// TwinCAT 3 PLC project Oefeningen3_
// ProgramVersion: 3.1.4024.0
// libraries:
//   Tc2_BABasic, * (Beckhoff Automation GmbH)
//   Tc2_Standard, * (Beckhoff Automation GmbH)
//   Tc2_System, * (Beckhoff Automation GmbH)
//   Tc2_Utilities, * (Beckhoff Automation GmbH)
//   Tc3_Module, * (Beckhoff Automation GmbH)
// project tree:
//   DUTs/ Pers_data.TcDUT
//   / GlobalTextList.TcGTLO, PlcTask.TcTTO, Visualization Manager.TcVMO (not stored)
//   POUs/ CheckBounds.TcPOU, CheckRangeInt.TcPOU, FB_Click_Log.TcPOU, FB_DrukknopSpecial.TcPOU, FB_GetMinimum.TcPOU, FB_PWM.TcPOU, FB_SearchString.TcPOU, FGetMinimum.TcPOU, MAIN.TcPOU, prg_Click_Log.TcPOU, prg_Druktoets_Functies.TcPOU, prg_GetMinimum.TcPOU, prg_Personeelsdata.TcPOU, prg_PWM.TcPOU, prg_SearchString.TcPOU
//   VISUs/ Visualization_Click_Logger.TcVIS, Visualization_GetMinimumClicker.TcVIS
// (motion and I/O tree: see PLC project oefeningen1)
// real-time tasks:
//   TASK PlcTask: cycle T#10ms, priority 20, ADS port 350
//   TASK PlcTask1: cycle T#10ms, priority 21, ADS port 351
//   TASK PlcTask2: cycle T#10ms, priority 22, ADS port 352
//   TASK PlcTask3: cycle T#10ms, priority 23, ADS port 353
//   TASK PlcTask4: cycle T#10ms, priority 24, ADS port 354

CONFIGURATION Oefeningen3_
    RESOURCE PLC ON TwinCAT3
        TASK PlcTask(INTERVAL := T#10ms, PRIORITY := 24);
        PROGRAM MAIN WITH PlcTask : MAIN;
    END_RESOURCE
END_CONFIGURATION

// ---- DUTs/Pers_data.TcDUT
TYPE Pers_data :
STRUCT
	Name      : STRING(25);
	Firstname : STRING(25);
	Age       : INT;
	Address   : STRING(55);
END_STRUCT
END_TYPE

// ---- POUs/MAIN.TcPOU
PROGRAM MAIN
VAR
END_VAR

//prg_PWM();
//prg_Click_Log();
//prg_GetMinimum();
//prg_Personeelsdata();
//prg_SearchString();
prg_Druktoets_Functies();

END_PROGRAM

// ---- POUs/prg_Druktoets_Functies.TcPOU
PROGRAM prg_Druktoets_Functies
VAR
	FB_Drukknop_Special: FB_DrukknopSpecial;
END_VAR

FB_Drukknop_Special(bDrukknop:= , bSingle=> , bDouble=> , bLong=> );

END_PROGRAM

// ---- POUs/FB_DrukknopSpecial.TcPOU
FUNCTION_BLOCK FB_DrukknopSpecial
VAR_INPUT
    bDrukknop : BOOL;          // fysiek knopsignaal
END_VAR

VAR_OUTPUT
    bSingle    : BOOL;
    bDouble    : BOOL;
    bLong      : BOOL;
END_VAR

VAR
    fbSD : FB_SingleDoubleClick;
    fbSL : FB_ShortLongClick;
END_VAR

// --- Doorgeven van de knop als input ---
fbSD(bSwitch := bDrukknop, tSwitchTime := T#500MS);
fbSL(bSwitch := bDrukknop, tSwitchTime := T#1S);

// --- Outputs ---
bSingle := fbSD.bSingleClick AND NOT fbSL.bLongClick;
bDouble := fbSD.bDoubleClick;
bLong   := fbSL.bLongClick;

END_FUNCTION_BLOCK

// ---- POUs/CheckBounds.TcPOU
FUNCTION CheckBounds : INT
VAR_INPUT
    InValue : INT;
END_VAR
VAR
END_VAR

IF InValue < 15 THEN
    CheckBounds := 15;
ELSIF InValue > 24 THEN
    CheckBounds := 24;
ELSE
    CheckBounds := InValue;
END_IF

END_FUNCTION

// ---- POUs/CheckRangeInt.TcPOU
FUNCTION CheckRangeInt : INT
VAR_INPUT
    InValue : INT;
END_VAR
VAR
END_VAR

IF InValue < 0 THEN
    CheckRangeInt := 0;
ELSIF InValue > 32767 THEN
    CheckRangeInt := 32767;
ELSE
    CheckRangeInt := InValue;
END_IF

END_FUNCTION

// ---- POUs/FB_Click_Log.TcPOU
FUNCTION_BLOCK FB_Click_Log
VAR_INPUT
    Drukknop    : BOOL;
END_VAR
VAR_OUTPUT
    Tijden      : ARRAY[1..10] OF TIME;
END_VAR
VAR
    tDrukRegistreren : TP;
    tPauze           : TP;
    FallingTimer     : F_TRIG;
    FallingPauze     : F_TRIG;

    RisingDruk       : R_TRIG;   
    Index            : INT := 0; 
    VorigeET         : TIME := T#0ms;   // nieuwe variabele om vorige tijd op te slaan
	i: INT;
END_VAR

(* Detecteer drukflank *)
RisingDruk(CLK := Drukknop);

(* 5s registratie *)
tDrukRegistreren(IN := Drukknop OR FallingPauze.Q, PT := T#5S);
FallingTimer(CLK := tDrukRegistreren.Q);

(* 2s pauze *)
tPauze(IN := FallingTimer.Q, PT := T#2S);
FallingPauze(CLK := tPauze.Q);

(* reset index na pauze *)
IF FallingPauze.Q THEN
    Index := 0;
    VorigeET := T#0MS;
	FOR i := 1 TO 10 DO
    Tijden[i] := T#0ms;
END_FOR;
END_IF

(* Registreer tijd bij elke drukflank *)
IF RisingDruk.Q AND tDrukRegistreren.Q THEN
    IF Index < 10 THEN
        Index := Index + 1;
        Tijden[Index] := tDrukRegistreren.ET - VorigeET;  // verschil tussen huidige en vorige druk
        VorigeET := tDrukRegistreren.ET;                  // update vorige tijd
    END_IF
END_IF

END_FUNCTION_BLOCK

// ---- POUs/FB_GetMinimum.TcPOU
FUNCTION_BLOCK FB_GetMinimum
VAR_INPUT
	Times : ARRAY[1..10] OF TIME;
END_VAR
VAR_OUTPUT
	MinTime : TIME;
END_VAR
VAR
	i : INT;
END_VAR

(* Initieel minimum = eerste element *)
MinTime := Times[1];

(* Vergelijk met rest van de array *)
FOR i := 2 TO 10 DO
	IF Times[i] < MinTime THEN
		MinTime := Times[i];
	END_IF
END_FOR;

END_FUNCTION_BLOCK

// ---- POUs/FB_PWM.TcPOU
FUNCTION_BLOCK FB_PWM
VAR_INPUT
    Enable     : BOOL;
    Periode    : TIME;   // totale PWM-periode
    DutyCycle  : INT;    // 0 .. 100 (%)
END_VAR

VAR_OUTPUT
    PWM_Out    : BOOL;
END_VAR

VAR
    tPWM       : TON;
    tOn        : TIME;
END_VAR

IF Enable THEN
    (* Bereken ON-tijd *)
    tOn := Periode * DutyCycle / 100;

    tPWM(IN := TRUE, PT := Periode);

    (* PWM-logica *)
    IF tPWM.ET < tOn THEN
        PWM_Out := TRUE;
    ELSE
        PWM_Out := FALSE;
    END_IF

    (* Periode herstarten *)
    IF tPWM.Q THEN
        tPWM(IN := FALSE);
    END_IF
ELSE
    PWM_Out := FALSE;
    tPWM(IN := FALSE);
END_IF

END_FUNCTION_BLOCK

// ---- POUs/FB_SearchString.TcPOU
FUNCTION_BLOCK FB_SearchString
VAR_INPUT
	Person    : Pers_data; //DUT STRUCT
	SearchTxt : STRING(25);
END_VAR
VAR_OUTPUT
	Match     : BOOL;
END_VAR
VAR
	AllText   : STRING(120);
	AllTextLower  : STRING(120);
	SearchLower   : STRING(25);
END_VAR

(* alles samenvoegen *)
AllText := CONCAT(
				CONCAT(Person.Name, Person.Firstname),
				Person.Address
			);

(* naar lowercase omzetten *)
AllTextLower := F_ToLCase(AllText);
SearchLower  := F_ToLCase(SearchTxt);

(* vergelijken *)
IF FIND(AllTextLower, SearchLower) > 0 THEN
	Match := TRUE;
ELSE
	Match := FALSE;
END_IF

END_FUNCTION_BLOCK

// ---- POUs/FGetMinimum.TcPOU
FUNCTION FGetMinimum : TIME
VAR_INPUT
	Times : ARRAY[1..10] OF TIME;
END_VAR
VAR
	i : INT;
	MinVal : TIME;
END_VAR

MinVal := Times[1];

FOR i := 2 TO 10 DO
	IF Times[i] < MinVal THEN
		MinVal := Times[i];
	END_IF
END_FOR;

FGetMinimum := MinVal;

END_FUNCTION

// ---- POUs/prg_Click_Log.TcPOU
PROGRAM prg_Click_Log
VAR	
	ClickLog: FB_Click_Log;

	bDrukknop		AT		%I*		:BOOL;
	LogTijden 		AT		%Q*		:ARRAY[1..10] OF TIME;
END_VAR

ClickLog(Drukknop:= bDrukknop, Tijden=> LogTijden);

END_PROGRAM

// ---- POUs/prg_GetMinimum.TcPOU
PROGRAM prg_GetMinimum
VAR
	FB_GetMinimum: FB_GetMinimum;
	FB_Click_Log: FB_Click_Log;
	bDrukknop		AT		%I*		:BOOL;
	tMinTime		AT		%Q*		:TIME;
	LogTijden 		:ARRAY[1..10] OF TIME;
END_VAR

FB_Click_Log(Drukknop:= bDrukknop, Tijden=> LogTijden);
FB_GetMinimum(Times:= LogTijden, MinTime=> tMinTime);

//Met een functie ipv FunctieBlok (ongetest)
//tMinTime := FGetMinimum(LogTijden);

END_PROGRAM

// ---- POUs/prg_Personeelsdata.TcPOU
PROGRAM prg_Personeelsdata
VAR
	Personeel : ARRAY[1..6] OF Pers_data;
END_VAR

(* P1 *)
Personeel[1].Name      := 'Müller';
Personeel[1].Firstname := 'Peter';
Personeel[1].Age       := 32;
Personeel[1].Address   := 'Postweg 34';

(* P2 *)
Personeel[2].Name      := 'Maesen';
Personeel[2].Firstname := 'Stijn';
Personeel[2].Age       := 15;
Personeel[2].Address   := 'Grote steenweg 8';

(* P3 *)
Personeel[3].Name      := 'Paque';
Personeel[3].Firstname := 'Stéphanie';
Personeel[3].Age       := 42;
Personeel[3].Address   := 'Tongersesteenweg 456';

(* P4 *)
Personeel[4].Name      := 'Fossen';
Personeel[4].Firstname := 'Jo';
Personeel[4].Age       := 20;
Personeel[4].Address   := 'Broekstraat 45';

(* P5 *)
Personeel[5].Name      := 'Poesmans';
Personeel[5].Firstname := 'Benny';
Personeel[5].Age       := 72;
Personeel[5].Address   := 'Veldweg 1A';

(* P6 *)
Personeel[6].Name      := 'Dybek';
Personeel[6].Firstname := 'Isolde';
Personeel[6].Age       := 55;
Personeel[6].Address   := 'Slagerijstraat 6';

END_PROGRAM

// ---- POUs/prg_PWM.TcPOU
PROGRAM prg_PWM
VAR
	PWM: FB_PWM;
	bPWMOUT		AT		%Q*		:BOOL;
END_VAR

PWM(Enable:= TRUE, Periode:= T#1S, DutyCycle:= 25, PWM_Out=> bPWMOUT);

END_PROGRAM

// ---- POUs/prg_SearchString.TcPOU
PROGRAM prg_SearchString
VAR
	Persoon : Pers_data := (
		Name := 'Peeters',
		Firstname := 'Stijn',
		Address := 'Kerkstraat 12'
	);

	SearchFB : FB_SearchString;
	Result   : BOOL;
END_VAR

SearchFB(
	Person := Persoon,
	SearchTxt := 'stijn'
);

Result := SearchFB.Match;

END_PROGRAM

// ---- GlobalTextList.TcGTLO
TEXTLIST GlobalTextList
  841 = 'Drukknop'
END_TEXTLIST

// ---- VISUs/Visualization_Click_Logger.TcVIS
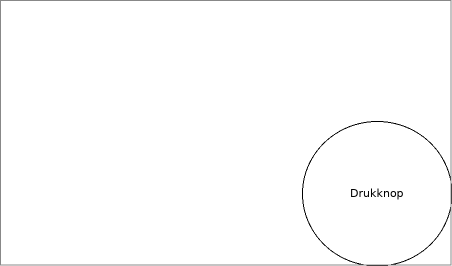
VISUALIZATION Visualization_Click_Logger  // 452x266
    Ellipse (302,121 150x145), "Drukknop"
        tap prg_GetMinimum.bDrukknop
END_VISUALIZATION

// ---- VISUs/Visualization_GetMinimumClicker.TcVIS
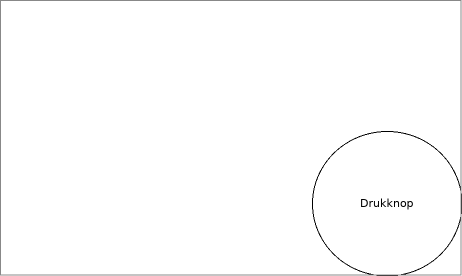
VISUALIZATION Visualization_GetMinimumClicker  // 462x276
    Ellipse (312,131 150x145), "Drukknop"
        tap prg_GetMinimum.bDrukknop
END_VISUALIZATION
